KUKA KRL program: kvp_lin.src, kvp_lin.dat

--- kvp_lin.src ---
&ACCESS RVP
&REL 16
&PARAM EDITMASK = *
&PARAM TEMPLATE = C:\KRC\Roboter\Template\vorgabe
DEF kvp_lin( )
;FOLD INI
  ;FOLD BASISTECH INI
    GLOBAL INTERRUPT DECL 3 WHEN $STOPMESS==TRUE DO IR_STOPM ( )
    INTERRUPT ON 3
    BAS (#INITMOV,0 )
  ;ENDFOLD (BASISTECH INI)
  ;FOLD USER INI
    ;Make your modifications here

  ;ENDFOLD (USER INI)
;ENDFOLD (INI)
BAS(#TOOL,2)

$ADVANCE = 1;
AXIS_SET = $AXIS_ACT
ERRCODE = 1
PTP $AXIS_ACT
LOOP

POSE_GOAL = FORWARD(AXIS_SET,ERRCODE)
LIN POSE_GOAL C_DIS

ENDLOOP
END

--- kvp_lin.dat ---
&ACCESS RVO
&REL 2
&PARAM EDITMASK = *
&PARAM TEMPLATE = C:\KRC\Roboter\Template\vorgabe
DEFDAT kvp_lin
;FOLD EXTERNAL DECLARATIONS;%{PE}%MKUKATPBASIS,%CEXT,%VCOMMON,%P
;FOLD BASISTECH EXT;%{PE}%MKUKATPBASIS,%CEXT,%VEXT,%P
EXT  BAS (BAS_COMMAND  :IN,REAL  :IN )
DECL INT SUCCESS
;ENDFOLD (BASISTECH EXT)
;FOLD USER EXT;%{E}%MKUKATPUSER,%CEXT,%VEXT,%P
;Make your modifications here

;ENDFOLD (USER EXT)
;ENDFOLD (EXTERNAL DECLARATIONS)
DECL E6AXIS AXIS_SET
DECL E6POS POSE_GOAL
DECL INT ERRCODE
ENDDAT
